FUNCTION_BLOCK FB_StateMachine
VAR_INPUT
END_VAR
VAR_OUTPUT
END_VAR
VAR
END_VAR

METHOD PROTECTED Fault
VAR_INPUT
END_VAR
END_METHOD

METHOD PROTECTED None
VAR_INPUT
END_VAR
END_METHOD

METHOD PROTECTED Ready
VAR_INPUT
END_VAR
END_METHOD

METHOD PROTECTED Running
VAR_INPUT
END_VAR
END_METHOD

METHOD PROTECTED Starting
VAR_INPUT
END_VAR
END_METHOD

METHOD PROTECTED Stopping
VAR_INPUT
END_VAR
END_METHOD

END_FUNCTION_BLOCK

(* stored: Version 1.1.0.1, ProductVersion 3.1.4024.10
   POU FB_StateMachine: Id {e7bd9ab3-42c4-4fd9-89cc-8e485c18b9aa}, SpecialFunc None
   Method Fault: Id {5403c10c-9f27-4105-9929-b3fdaebab555}
   Method None: Id {c26a898b-4759-4bf0-9a7e-4fbed4a3aa71}
   Method Ready: Id {733a1433-3fcd-405d-ae59-5126c28fe665}
   Method Running: Id {19f67fcc-a3e9-4f75-a7ef-2c803bfa74f5}
   Method Starting: Id {18f478f5-7418-40e6-8d07-83064c9734d7}
   Method Stopping: Id {5a0ad9fe-8672-4d85-b78b-f34822a45ee6} *)
